(* Logix 5000 project; controller NSH_PLC1 vendor 1 type 14 code 167 rev 32.11; software revision 32.02; part 4 of 12 *)
(* tags used below, declared in another part *)
   H42C : Motor;   // S.Roll
   H42D : Motor;   // Shr.Roll.
   H43A : Motor;   // Aspirator
   H43B : Motor;   // Aspirator
   H49 : Motor;   // Ele.
   H50A : Motor;   // Auger
   H50B : Motor;   // Auger
   M16 : Motor;   // Evo.
   M17 : Motor;   // Evo.
   M18 : Motor;   // Vib.
   M19 : Motor;   // Ele.
   S1 : Motor;   // Vib.
   S10 : Motor;   // Auger
   S13 : Motor;   // Ele.
   S14 : Motor;   // Auger
   S15 : Motor;   // Auger
   S16A : Motor;   // Auger
   S16B : Motor;   // Auger
   S17A : Motor;   // HS Cracker
   S17B : Motor;   // Hard Crkr.
   S17C : Motor;   // Shr.Roll.
   S17D : Motor;   // S.Roll
   S18A : Motor;   // HC Vib.
   S18B : Motor;   // Hard Crkr.
   S18C : Motor;   // Shr.Roll.
   S18D : Motor;   // S.Roll
   S19 : Motor;   // Gry.
   S2 : Motor;   // Ele.
   S20 : Motor;   // Ele.
   S21 : Motor;   // Roll Fdr.
   S22A : Motor;   // HC Vib.
   S22B : Motor;   // Hard Crkr.
   S22C : Motor;   // Shr.Roll.
   S22D : Motor;   // S.Roll
   S23A : Motor;   // HC Vib.
   S23B : Motor;   // Hard Crkr.
   S23C : Motor;   // Shr.Roll.
   S23D : Motor;   // S.Roll
   S24 : Motor;   // Deck
   S25 : Motor;   // Ele.
   S26 : Motor;   // Auger
   S27 : Motor;   // Roll Fdr
   S28A : Motor;   // HC Vib.
   S28B : Motor;   // Hard Crkr.
   S28C : Motor;   // Shr.Roll.
   S28D : Motor;   // S.Roll
   S29A : Motor;   // HC Vib.
   S29B : Motor;   // Hard Crkr.
   S29C : Motor;   // Shr.Roll.
   S29D : Motor;   // S.Roll
   S3 : Motor;   // Auger
   S30 : Motor;   // Ele.
   S31 : Motor;   // Auger
   S32A : Motor;   // HC Vib.
   S32B : Motor;   // Hard Crkr.
   S34 : Motor;   // Deck
   S35 : Motor;   // Ele.
   S36 : Motor;   // Auger
   S38 : Motor;   // Shkr.
   S39 : Motor;   // Ele.
   S41 : Motor;   // Ele.
   S43 : Motor;   // Shkr.
   S44 : Motor;   // Ele.
   S45 : Motor;   // Auger
   S4A : Motor;   // Aspirator
   S4B : Motor;   // Aspirator
   S5A : Motor;   // Aspirator
   S5B : Motor;   // Aspirator
   S6 : Motor;   // Belt
   S7 : Motor;   // Ele.
   S8 : Motor;   // Auger
   S9 : Motor;   // Ele.
(* HullerSheller, continued *)

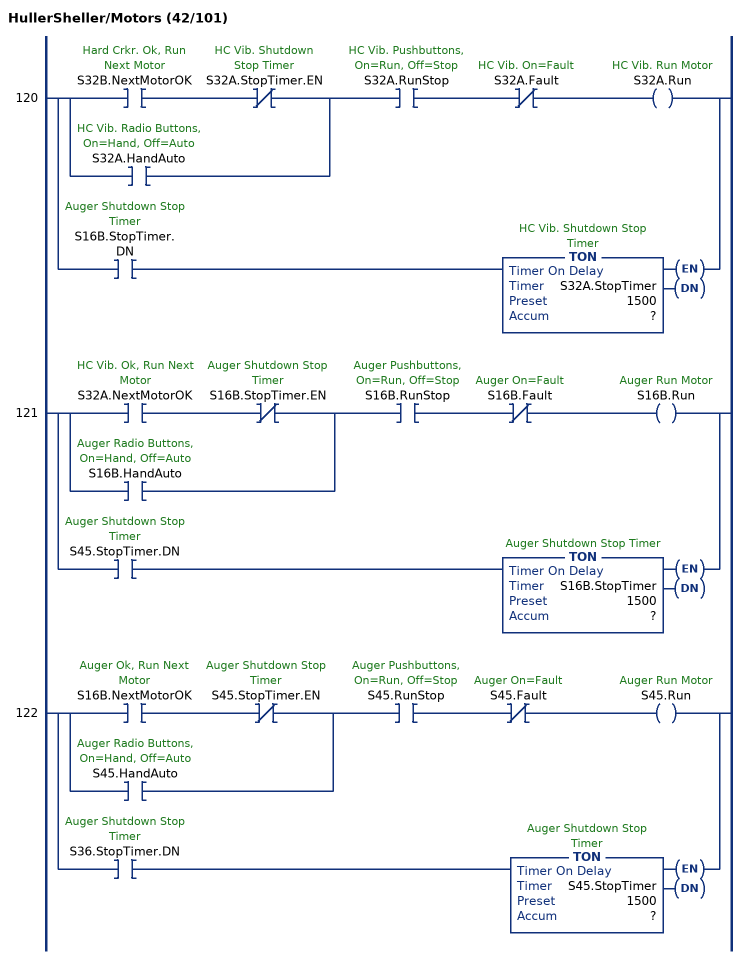
   [picture p66: HullerSheller/Motors rungs 120-122]
   120: [[XIC(S32B.NextMotorOK) XIO(S32A.StopTimer.EN) ,XIC(S32A.HandAuto) ] XIC(S32A.RunStop) XIO(S32A.Fault) OTE(S32A.Run) ,XIC(S16B.StopTimer.DN) TON(S32A.StopTimer,?,?) ];
   121: [[XIC(S32A.NextMotorOK) XIO(S16B.StopTimer.EN) ,XIC(S16B.HandAuto) ] XIC(S16B.RunStop) XIO(S16B.Fault) OTE(S16B.Run) ,XIC(S45.StopTimer.DN) TON(S16B.StopTimer,?,?) ];
   122: [[XIC(S16B.NextMotorOK) XIO(S45.StopTimer.EN) ,XIC(S45.HandAuto) ] XIC(S45.RunStop) XIO(S45.Fault) OTE(S45.Run) ,XIC(S36.StopTimer.DN) TON(S45.StopTimer,?,?) ];
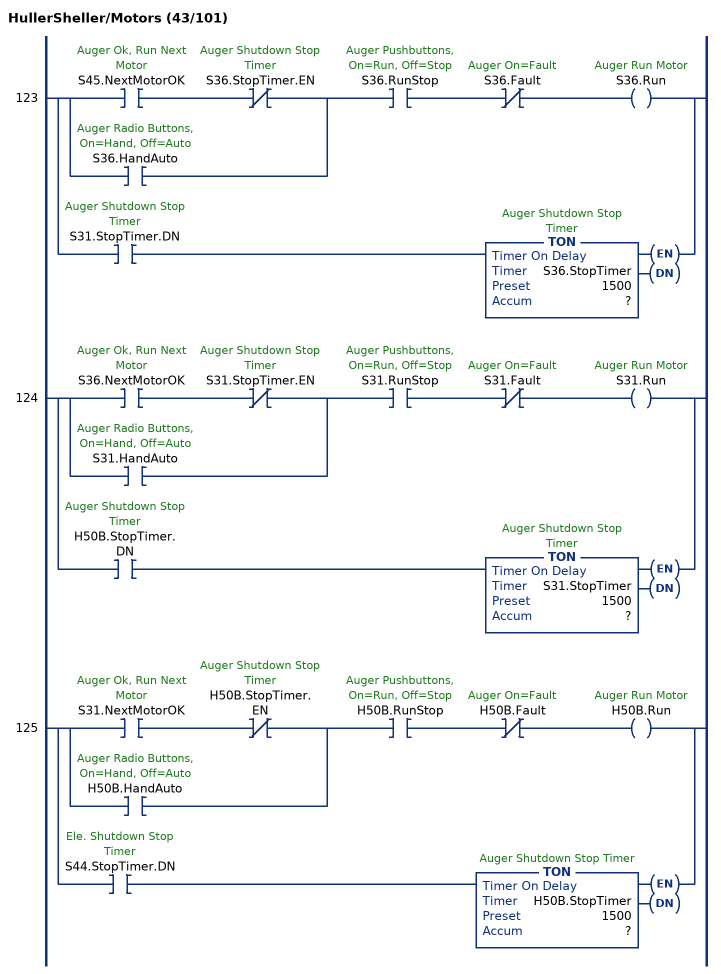
   123: [[XIC(S45.NextMotorOK) XIO(S36.StopTimer.EN) ,XIC(S36.HandAuto) ] XIC(S36.RunStop) XIO(S36.Fault) OTE(S36.Run) ,XIC(S31.StopTimer.DN) TON(S36.StopTimer,?,?) ];
   124: [[XIC(S36.NextMotorOK) XIO(S31.StopTimer.EN) ,XIC(S31.HandAuto) ] XIC(S31.RunStop) XIO(S31.Fault) OTE(S31.Run) ,XIC(H50B.StopTimer.DN) TON(S31.StopTimer,?,?) ];
   125: [[XIC(S31.NextMotorOK) XIO(H50B.StopTimer.EN) ,XIC(H50B.HandAuto) ] XIC(H50B.RunStop) XIO(H50B.Fault) OTE(H50B.Run) ,XIC(S44.StopTimer.DN) TON(H50B.StopTimer,?,?) ];
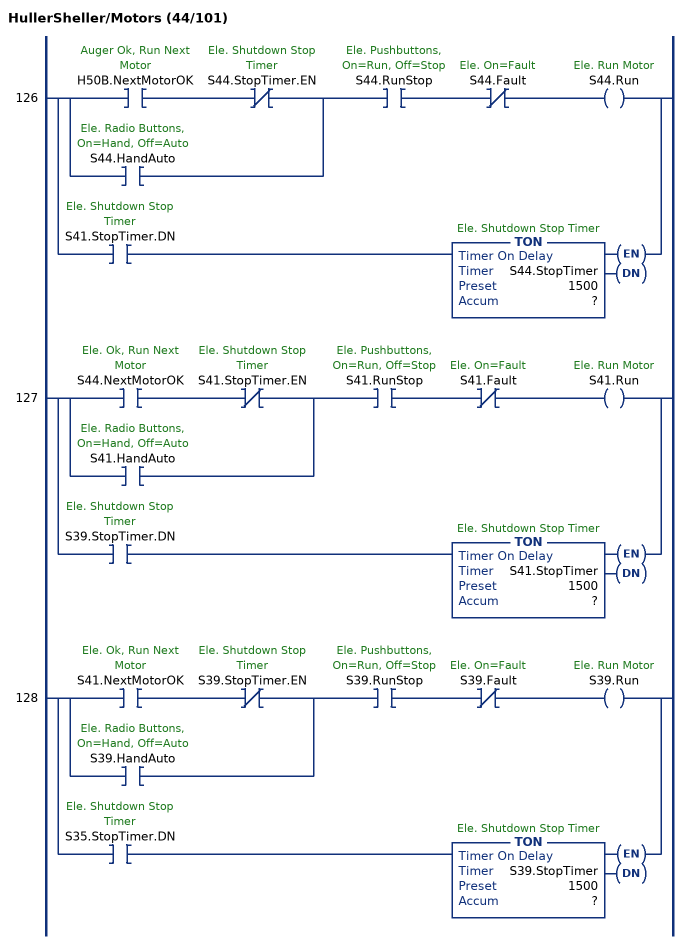
   126: [[XIC(H50B.NextMotorOK) XIO(S44.StopTimer.EN) ,XIC(S44.HandAuto) ] XIC(S44.RunStop) XIO(S44.Fault) OTE(S44.Run) ,XIC(S41.StopTimer.DN) TON(S44.StopTimer,?,?) ];
   127: [[XIC(S44.NextMotorOK) XIO(S41.StopTimer.EN) ,XIC(S41.HandAuto) ] XIC(S41.RunStop) XIO(S41.Fault) OTE(S41.Run) ,XIC(S39.StopTimer.DN) TON(S41.StopTimer,?,?) ];
   128: [[XIC(S41.NextMotorOK) XIO(S39.StopTimer.EN) ,XIC(S39.HandAuto) ] XIC(S39.RunStop) XIO(S39.Fault) OTE(S39.Run) ,XIC(S35.StopTimer.DN) TON(S39.StopTimer,?,?) ];
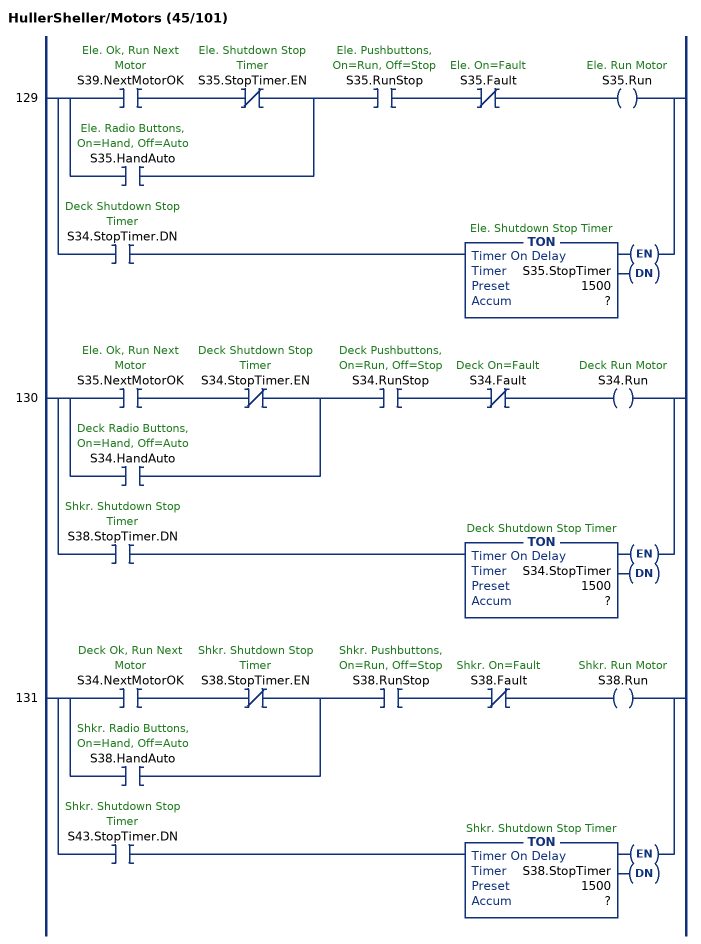
   129: [[XIC(S39.NextMotorOK) XIO(S35.StopTimer.EN) ,XIC(S35.HandAuto) ] XIC(S35.RunStop) XIO(S35.Fault) OTE(S35.Run) ,XIC(S34.StopTimer.DN) TON(S35.StopTimer,?,?) ];
   130: [[XIC(S35.NextMotorOK) XIO(S34.StopTimer.EN) ,XIC(S34.HandAuto) ] XIC(S34.RunStop) XIO(S34.Fault) OTE(S34.Run) ,XIC(S38.StopTimer.DN) TON(S34.StopTimer,?,?) ];
   131: [[XIC(S34.NextMotorOK) XIO(S38.StopTimer.EN) ,XIC(S38.HandAuto) ] XIC(S38.RunStop) XIO(S38.Fault) OTE(S38.Run) ,XIC(S43.StopTimer.DN) TON(S38.StopTimer,?,?) ];
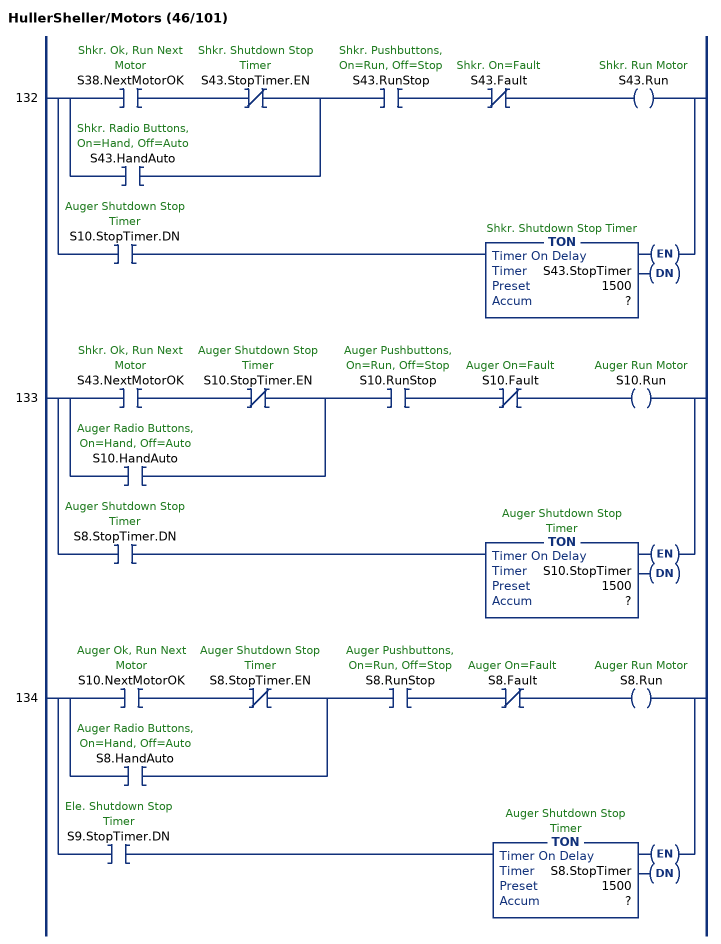
   132: [[XIC(S38.NextMotorOK) XIO(S43.StopTimer.EN) ,XIC(S43.HandAuto) ] XIC(S43.RunStop) XIO(S43.Fault) OTE(S43.Run) ,XIC(S10.StopTimer.DN) TON(S43.StopTimer,?,?) ];
   133: [[XIC(S43.NextMotorOK) XIO(S10.StopTimer.EN) ,XIC(S10.HandAuto) ] XIC(S10.RunStop) XIO(S10.Fault) OTE(S10.Run) ,XIC(S8.StopTimer.DN) TON(S10.StopTimer,?,?) ];
   134: [[XIC(S10.NextMotorOK) XIO(S8.StopTimer.EN) ,XIC(S8.HandAuto) ] XIC(S8.RunStop) XIO(S8.Fault) OTE(S8.Run) ,XIC(S9.StopTimer.DN) TON(S8.StopTimer,?,?) ];
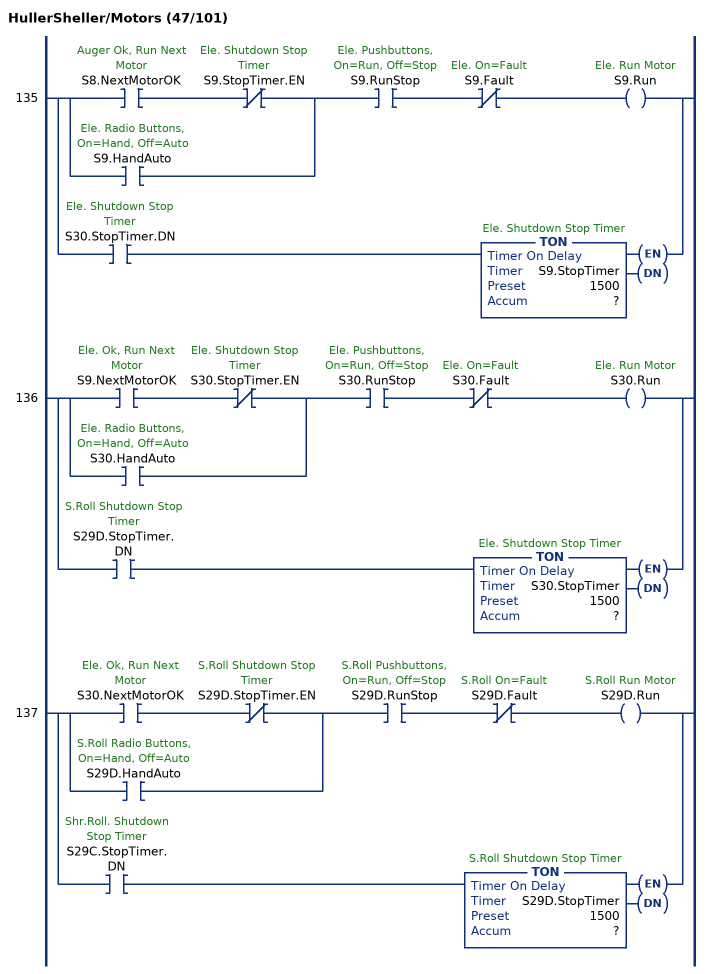
   135: [[XIC(S8.NextMotorOK) XIO(S9.StopTimer.EN) ,XIC(S9.HandAuto) ] XIC(S9.RunStop) XIO(S9.Fault) OTE(S9.Run) ,XIC(S30.StopTimer.DN) TON(S9.StopTimer,?,?) ];
   136: [[XIC(S9.NextMotorOK) XIO(S30.StopTimer.EN) ,XIC(S30.HandAuto) ] XIC(S30.RunStop) XIO(S30.Fault) OTE(S30.Run) ,XIC(S29D.StopTimer.DN) TON(S30.StopTimer,?,?) ];
   137: [[XIC(S30.NextMotorOK) XIO(S29D.StopTimer.EN) ,XIC(S29D.HandAuto) ] XIC(S29D.RunStop) XIO(S29D.Fault) OTE(S29D.Run) ,XIC(S29C.StopTimer.DN) TON(S29D.StopTimer,?,?) ];
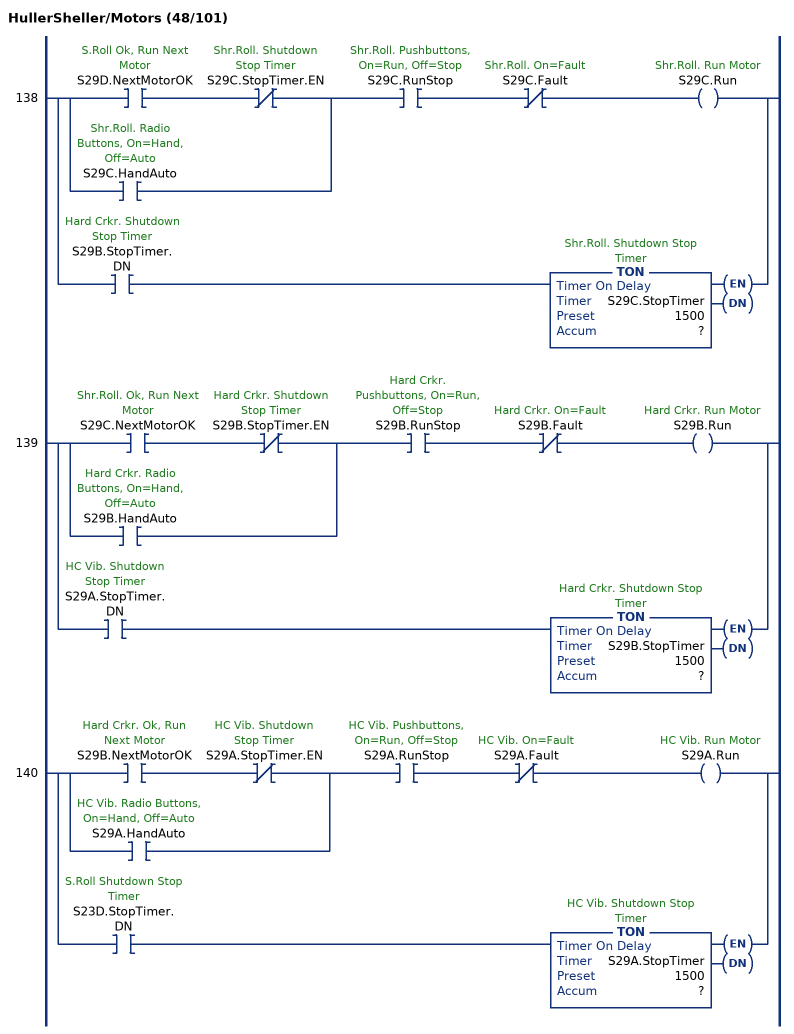
   138: [[XIC(S29D.NextMotorOK) XIO(S29C.StopTimer.EN) ,XIC(S29C.HandAuto) ] XIC(S29C.RunStop) XIO(S29C.Fault) OTE(S29C.Run) ,XIC(S29B.StopTimer.DN) TON(S29C.StopTimer,?,?) ];
   139: [[XIC(S29C.NextMotorOK) XIO(S29B.StopTimer.EN) ,XIC(S29B.HandAuto) ] XIC(S29B.RunStop) XIO(S29B.Fault) OTE(S29B.Run) ,XIC(S29A.StopTimer.DN) TON(S29B.StopTimer,?,?) ];
   140: [[XIC(S29B.NextMotorOK) XIO(S29A.StopTimer.EN) ,XIC(S29A.HandAuto) ] XIC(S29A.RunStop) XIO(S29A.Fault) OTE(S29A.Run) ,XIC(S23D.StopTimer.DN) TON(S29A.StopTimer,?,?) ];
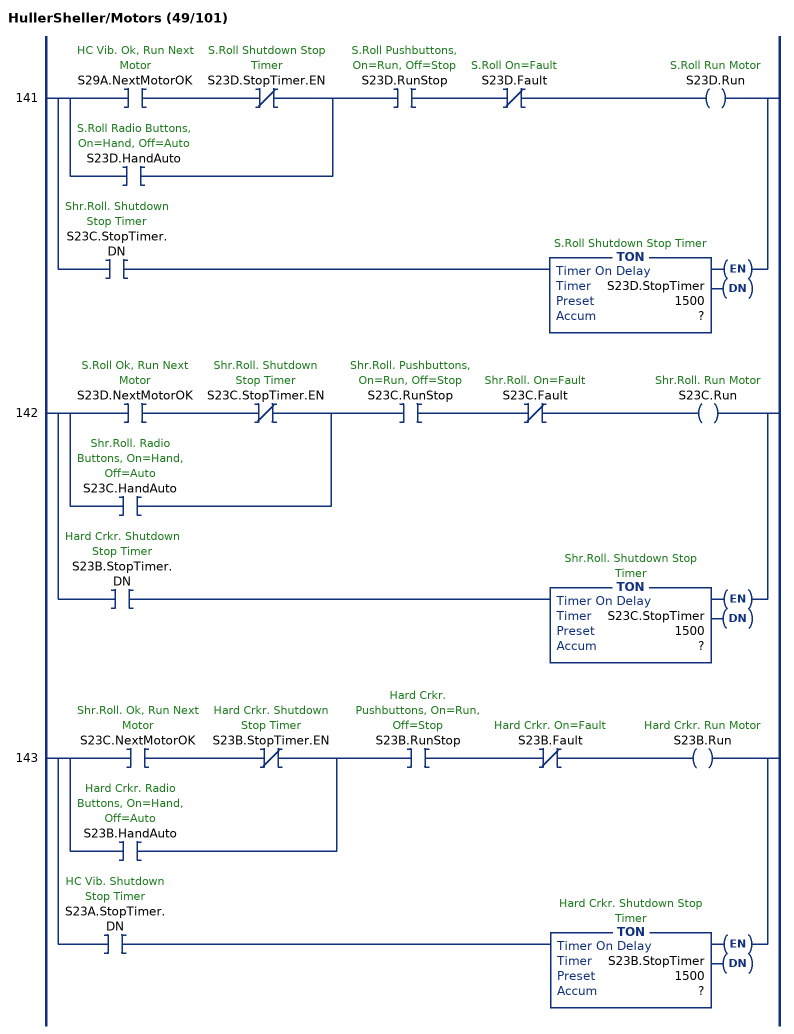
   141: [[XIC(S29A.NextMotorOK) XIO(S23D.StopTimer.EN) ,XIC(S23D.HandAuto) ] XIC(S23D.RunStop) XIO(S23D.Fault) OTE(S23D.Run) ,XIC(S23C.StopTimer.DN) TON(S23D.StopTimer,?,?) ];
   142: [[XIC(S23D.NextMotorOK) XIO(S23C.StopTimer.EN) ,XIC(S23C.HandAuto) ] XIC(S23C.RunStop) XIO(S23C.Fault) OTE(S23C.Run) ,XIC(S23B.StopTimer.DN) TON(S23C.StopTimer,?,?) ];
   143: [[XIC(S23C.NextMotorOK) XIO(S23B.StopTimer.EN) ,XIC(S23B.HandAuto) ] XIC(S23B.RunStop) XIO(S23B.Fault) OTE(S23B.Run) ,XIC(S23A.StopTimer.DN) TON(S23B.StopTimer,?,?) ];
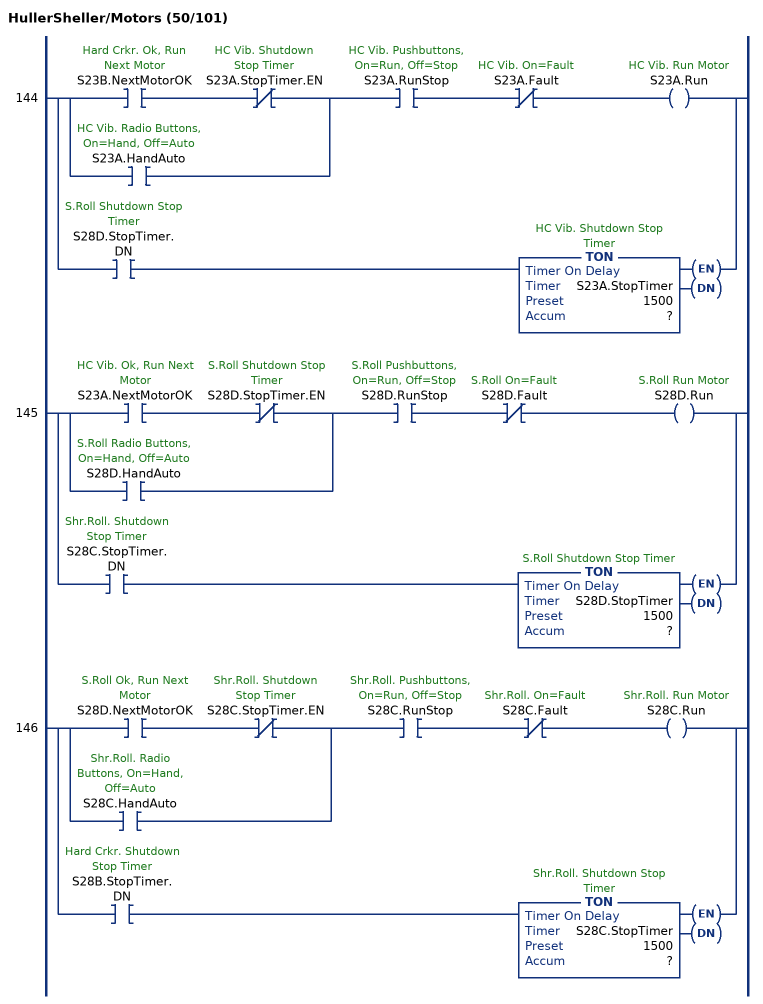
   144: [[XIC(S23B.NextMotorOK) XIO(S23A.StopTimer.EN) ,XIC(S23A.HandAuto) ] XIC(S23A.RunStop) XIO(S23A.Fault) OTE(S23A.Run) ,XIC(S28D.StopTimer.DN) TON(S23A.StopTimer,?,?) ];
   145: [[XIC(S23A.NextMotorOK) XIO(S28D.StopTimer.EN) ,XIC(S28D.HandAuto) ] XIC(S28D.RunStop) XIO(S28D.Fault) OTE(S28D.Run) ,XIC(S28C.StopTimer.DN) TON(S28D.StopTimer,?,?) ];
   146: [[XIC(S28D.NextMotorOK) XIO(S28C.StopTimer.EN) ,XIC(S28C.HandAuto) ] XIC(S28C.RunStop) XIO(S28C.Fault) OTE(S28C.Run) ,XIC(S28B.StopTimer.DN) TON(S28C.StopTimer,?,?) ];
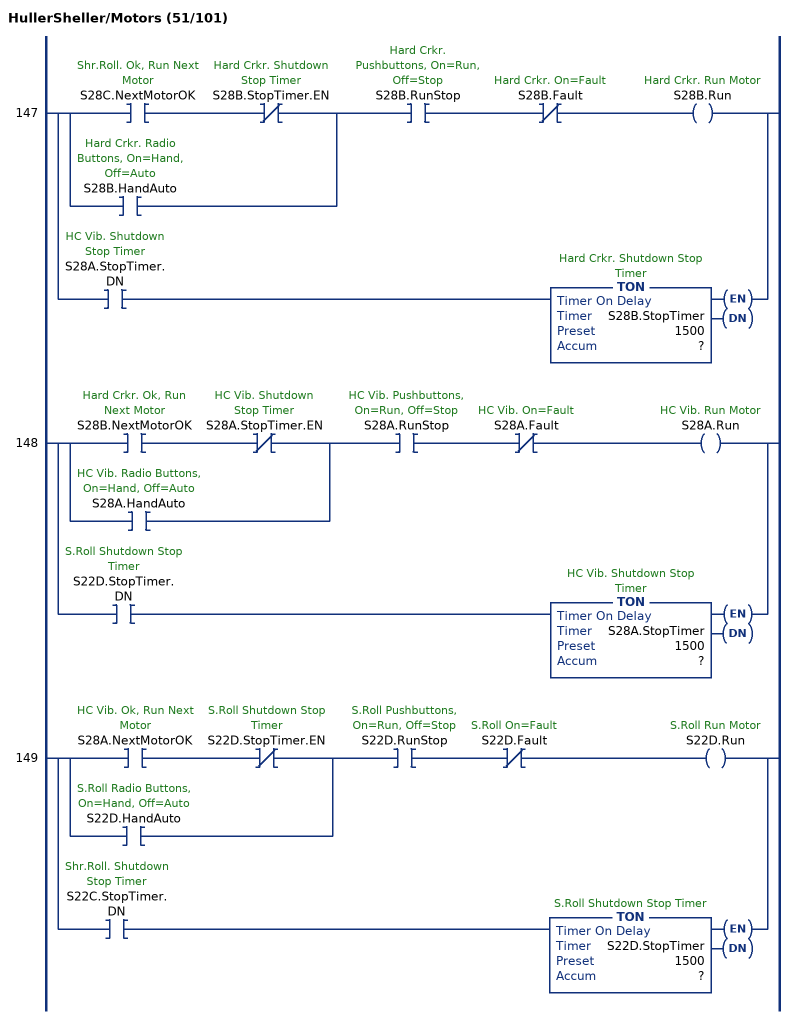
   147: [[XIC(S28C.NextMotorOK) XIO(S28B.StopTimer.EN) ,XIC(S28B.HandAuto) ] XIC(S28B.RunStop) XIO(S28B.Fault) OTE(S28B.Run) ,XIC(S28A.StopTimer.DN) TON(S28B.StopTimer,?,?) ];
   148: [[XIC(S28B.NextMotorOK) XIO(S28A.StopTimer.EN) ,XIC(S28A.HandAuto) ] XIC(S28A.RunStop) XIO(S28A.Fault) OTE(S28A.Run) ,XIC(S22D.StopTimer.DN) TON(S28A.StopTimer,?,?) ];
   149: [[XIC(S28A.NextMotorOK) XIO(S22D.StopTimer.EN) ,XIC(S22D.HandAuto) ] XIC(S22D.RunStop) XIO(S22D.Fault) OTE(S22D.Run) ,XIC(S22C.StopTimer.DN) TON(S22D.StopTimer,?,?) ];
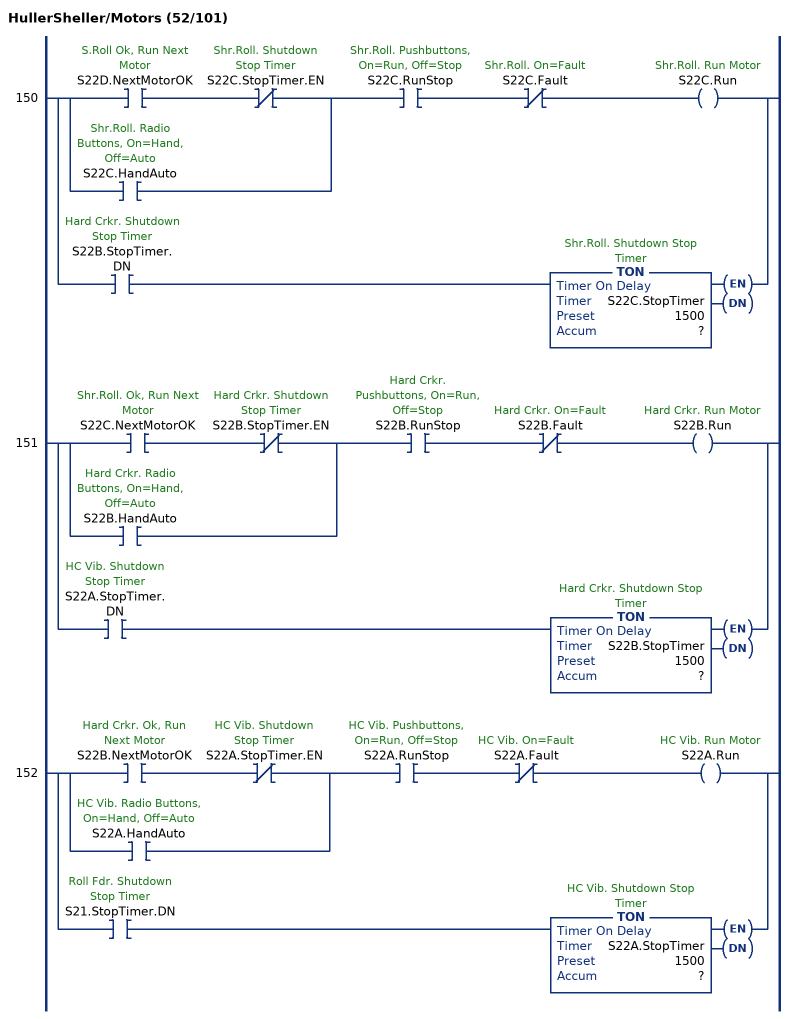
   150: [[XIC(S22D.NextMotorOK) XIO(S22C.StopTimer.EN) ,XIC(S22C.HandAuto) ] XIC(S22C.RunStop) XIO(S22C.Fault) OTE(S22C.Run) ,XIC(S22B.StopTimer.DN) TON(S22C.StopTimer,?,?) ];
   151: [[XIC(S22C.NextMotorOK) XIO(S22B.StopTimer.EN) ,XIC(S22B.HandAuto) ] XIC(S22B.RunStop) XIO(S22B.Fault) OTE(S22B.Run) ,XIC(S22A.StopTimer.DN) TON(S22B.StopTimer,?,?) ];
   152: [[XIC(S22B.NextMotorOK) XIO(S22A.StopTimer.EN) ,XIC(S22A.HandAuto) ] XIC(S22A.RunStop) XIO(S22A.Fault) OTE(S22A.Run) ,XIC(S21.StopTimer.DN) TON(S22A.StopTimer,?,?) ];
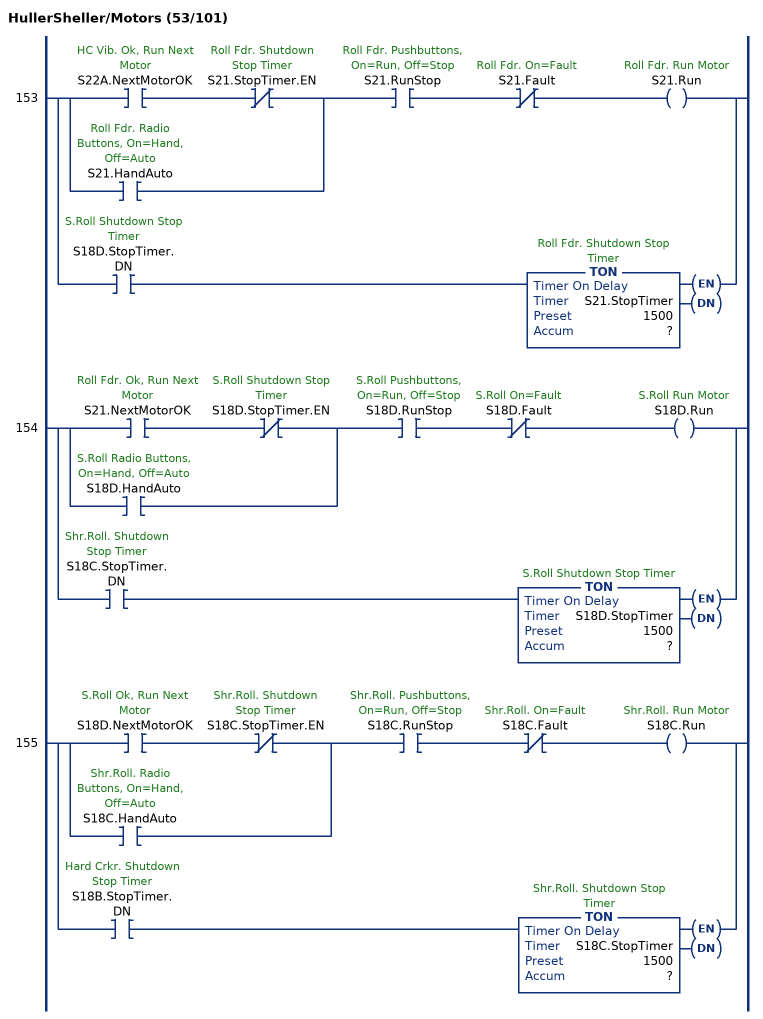
   153: [[XIC(S22A.NextMotorOK) XIO(S21.StopTimer.EN) ,XIC(S21.HandAuto) ] XIC(S21.RunStop) XIO(S21.Fault) OTE(S21.Run) ,XIC(S18D.StopTimer.DN) TON(S21.StopTimer,?,?) ];
   154: [[XIC(S21.NextMotorOK) XIO(S18D.StopTimer.EN) ,XIC(S18D.HandAuto) ] XIC(S18D.RunStop) XIO(S18D.Fault) OTE(S18D.Run) ,XIC(S18C.StopTimer.DN) TON(S18D.StopTimer,?,?) ];
   155: [[XIC(S18D.NextMotorOK) XIO(S18C.StopTimer.EN) ,XIC(S18C.HandAuto) ] XIC(S18C.RunStop) XIO(S18C.Fault) OTE(S18C.Run) ,XIC(S18B.StopTimer.DN) TON(S18C.StopTimer,?,?) ];
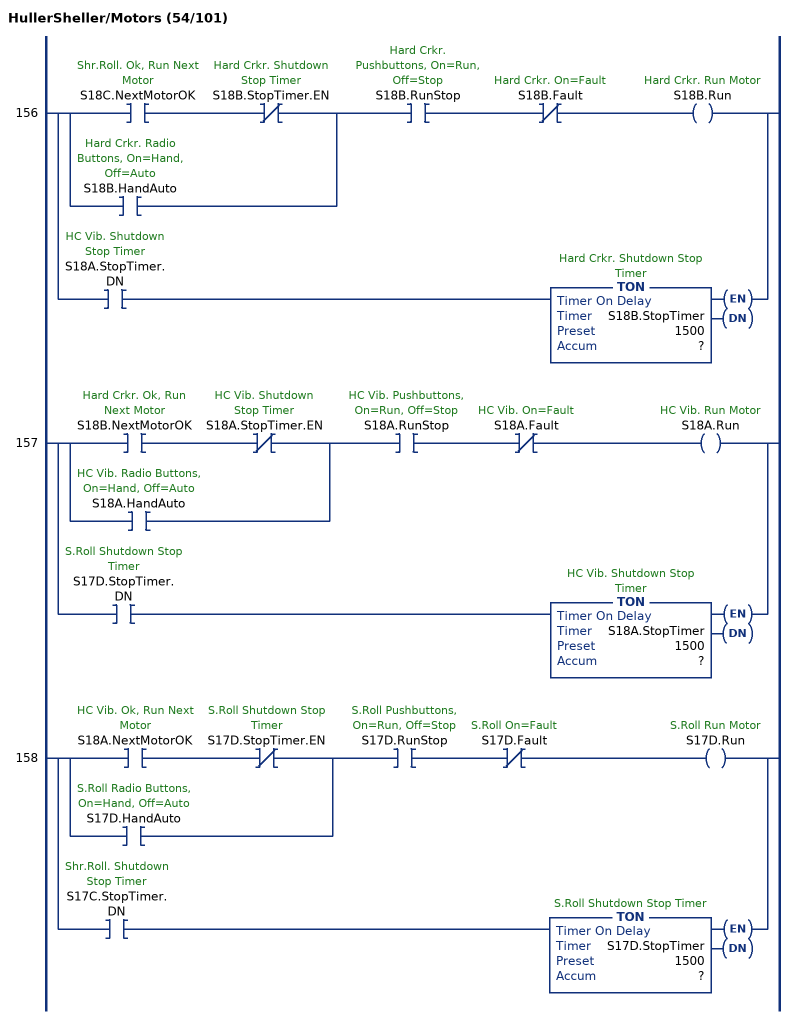
   156: [[XIC(S18C.NextMotorOK) XIO(S18B.StopTimer.EN) ,XIC(S18B.HandAuto) ] XIC(S18B.RunStop) XIO(S18B.Fault) OTE(S18B.Run) ,XIC(S18A.StopTimer.DN) TON(S18B.StopTimer,?,?) ];
   157: [[XIC(S18B.NextMotorOK) XIO(S18A.StopTimer.EN) ,XIC(S18A.HandAuto) ] XIC(S18A.RunStop) XIO(S18A.Fault) OTE(S18A.Run) ,XIC(S17D.StopTimer.DN) TON(S18A.StopTimer,?,?) ];
   158: [[XIC(S18A.NextMotorOK) XIO(S17D.StopTimer.EN) ,XIC(S17D.HandAuto) ] XIC(S17D.RunStop) XIO(S17D.Fault) OTE(S17D.Run) ,XIC(S17C.StopTimer.DN) TON(S17D.StopTimer,?,?) ];
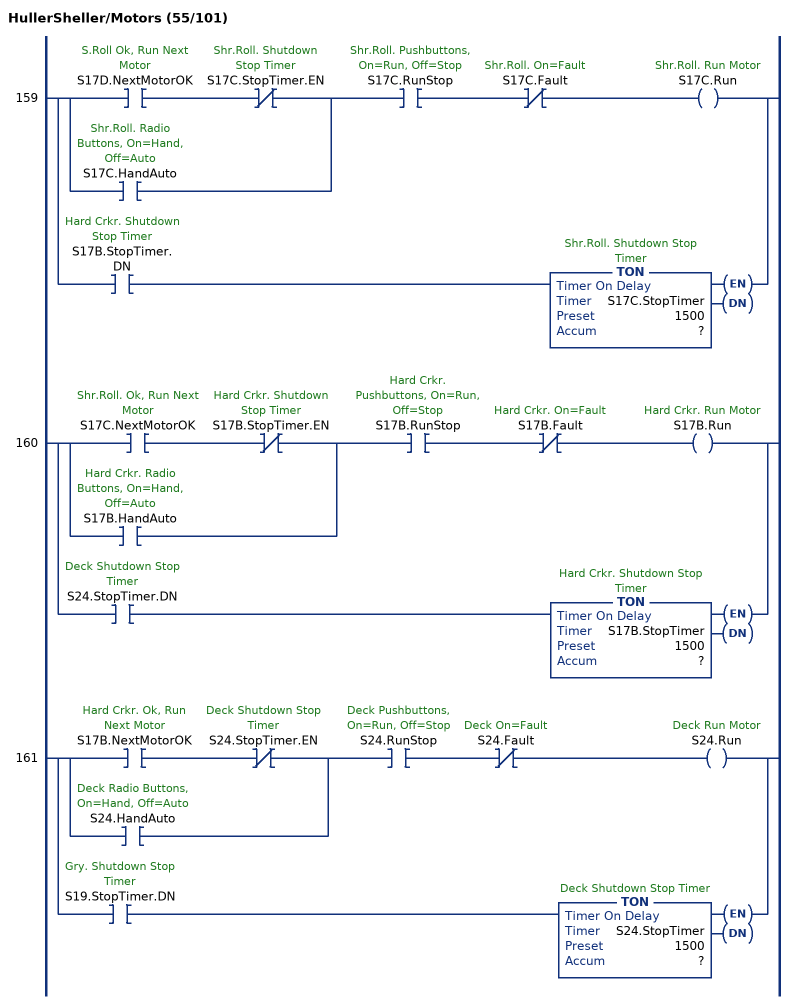
   159: [[XIC(S17D.NextMotorOK) XIO(S17C.StopTimer.EN) ,XIC(S17C.HandAuto) ] XIC(S17C.RunStop) XIO(S17C.Fault) OTE(S17C.Run) ,XIC(S17B.StopTimer.DN) TON(S17C.StopTimer,?,?) ];
   160: [[XIC(S17C.NextMotorOK) XIO(S17B.StopTimer.EN) ,XIC(S17B.HandAuto) ] XIC(S17B.RunStop) XIO(S17B.Fault) OTE(S17B.Run) ,XIC(S24.StopTimer.DN) TON(S17B.StopTimer,?,?) ];
   161: [[XIC(S17B.NextMotorOK) XIO(S24.StopTimer.EN) ,XIC(S24.HandAuto) ] XIC(S24.RunStop) XIO(S24.Fault) OTE(S24.Run) ,XIC(S19.StopTimer.DN) TON(S24.StopTimer,?,?) ];
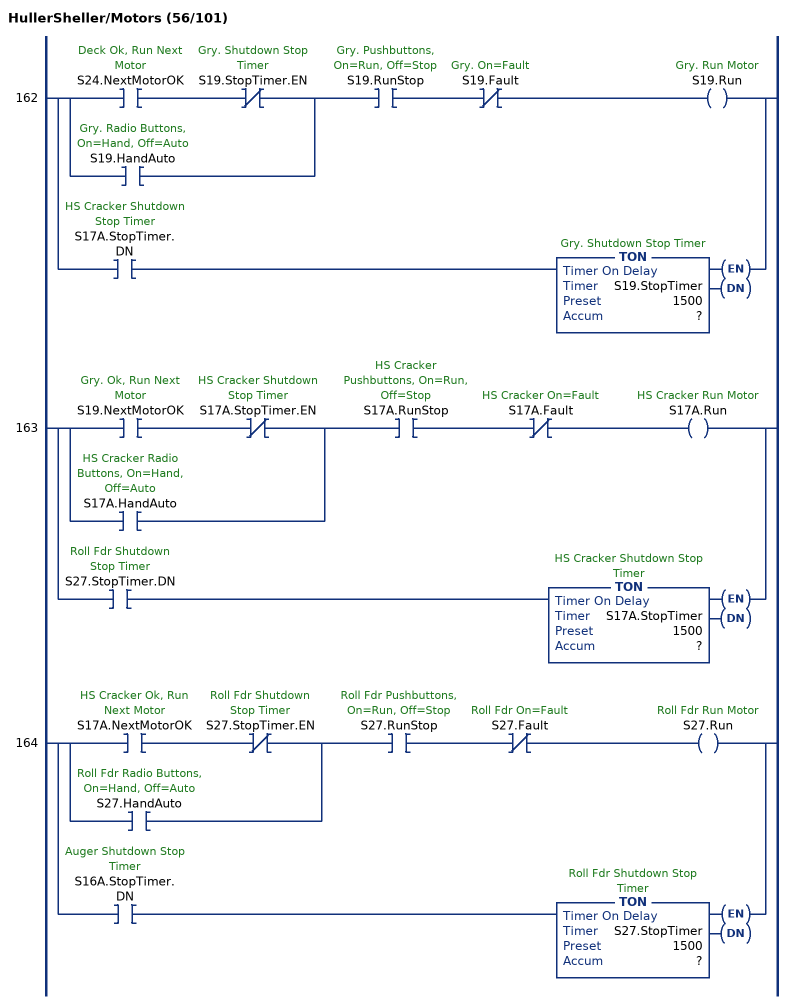
   162: [[XIC(S24.NextMotorOK) XIO(S19.StopTimer.EN) ,XIC(S19.HandAuto) ] XIC(S19.RunStop) XIO(S19.Fault) OTE(S19.Run) ,XIC(S17A.StopTimer.DN) TON(S19.StopTimer,?,?) ];
   163: [[XIC(S19.NextMotorOK) XIO(S17A.StopTimer.EN) ,XIC(S17A.HandAuto) ] XIC(S17A.RunStop) XIO(S17A.Fault) OTE(S17A.Run) ,XIC(S27.StopTimer.DN) TON(S17A.StopTimer,?,?) ];
   164: [[XIC(S17A.NextMotorOK) XIO(S27.StopTimer.EN) ,XIC(S27.HandAuto) ] XIC(S27.RunStop) XIO(S27.Fault) OTE(S27.Run) ,XIC(S16A.StopTimer.DN) TON(S27.StopTimer,?,?) ];
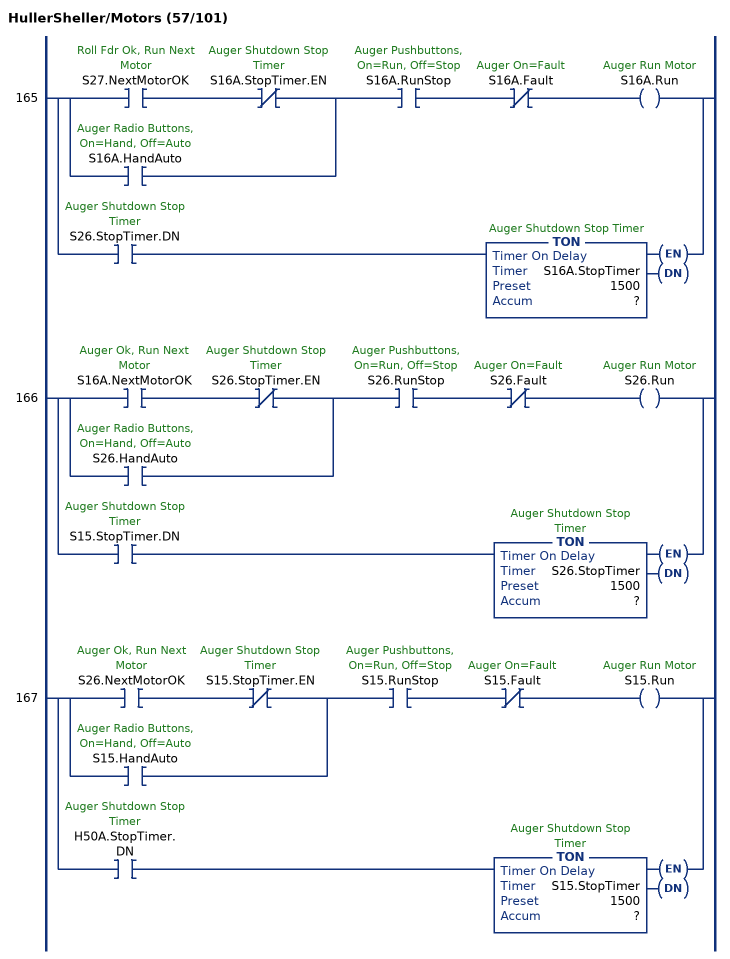
   165: [[XIC(S27.NextMotorOK) XIO(S16A.StopTimer.EN) ,XIC(S16A.HandAuto) ] XIC(S16A.RunStop) XIO(S16A.Fault) OTE(S16A.Run) ,XIC(S26.StopTimer.DN) TON(S16A.StopTimer,?,?) ];
   166: [[XIC(S16A.NextMotorOK) XIO(S26.StopTimer.EN) ,XIC(S26.HandAuto) ] XIC(S26.RunStop) XIO(S26.Fault) OTE(S26.Run) ,XIC(S15.StopTimer.DN) TON(S26.StopTimer,?,?) ];
   167: [[XIC(S26.NextMotorOK) XIO(S15.StopTimer.EN) ,XIC(S15.HandAuto) ] XIC(S15.RunStop) XIO(S15.Fault) OTE(S15.Run) ,XIC(H50A.StopTimer.DN) TON(S15.StopTimer,?,?) ];
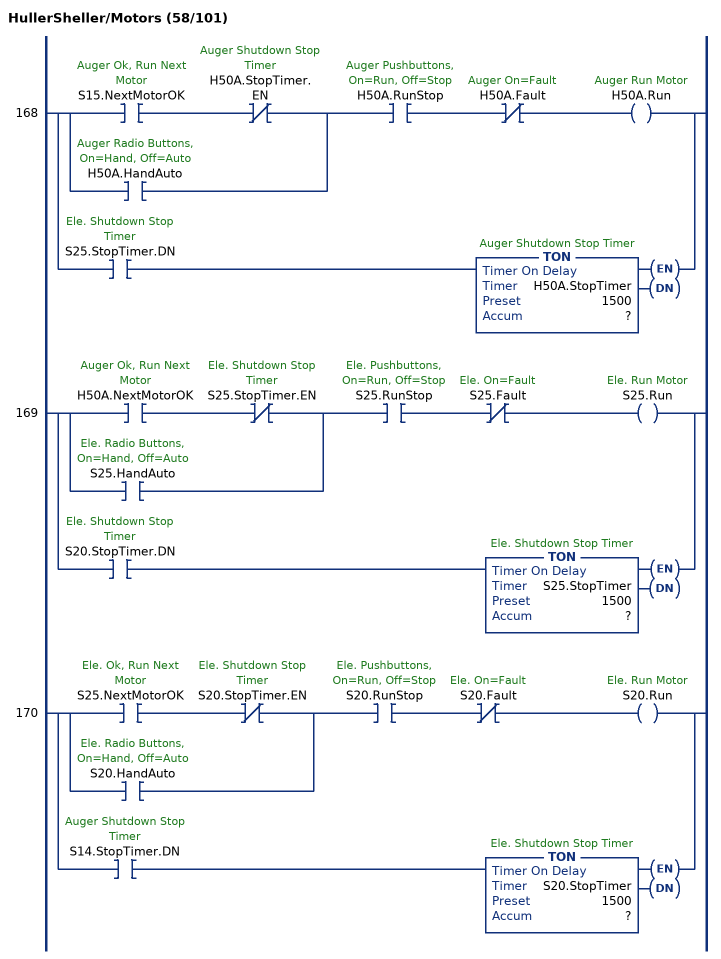
   168: [[XIC(S15.NextMotorOK) XIO(H50A.StopTimer.EN) ,XIC(H50A.HandAuto) ] XIC(H50A.RunStop) XIO(H50A.Fault) OTE(H50A.Run) ,XIC(S25.StopTimer.DN) TON(H50A.StopTimer,?,?) ];
   169: [[XIC(H50A.NextMotorOK) XIO(S25.StopTimer.EN) ,XIC(S25.HandAuto) ] XIC(S25.RunStop) XIO(S25.Fault) OTE(S25.Run) ,XIC(S20.StopTimer.DN) TON(S25.StopTimer,?,?) ];
   170: [[XIC(S25.NextMotorOK) XIO(S20.StopTimer.EN) ,XIC(S20.HandAuto) ] XIC(S20.RunStop) XIO(S20.Fault) OTE(S20.Run) ,XIC(S14.StopTimer.DN) TON(S20.StopTimer,?,?) ];
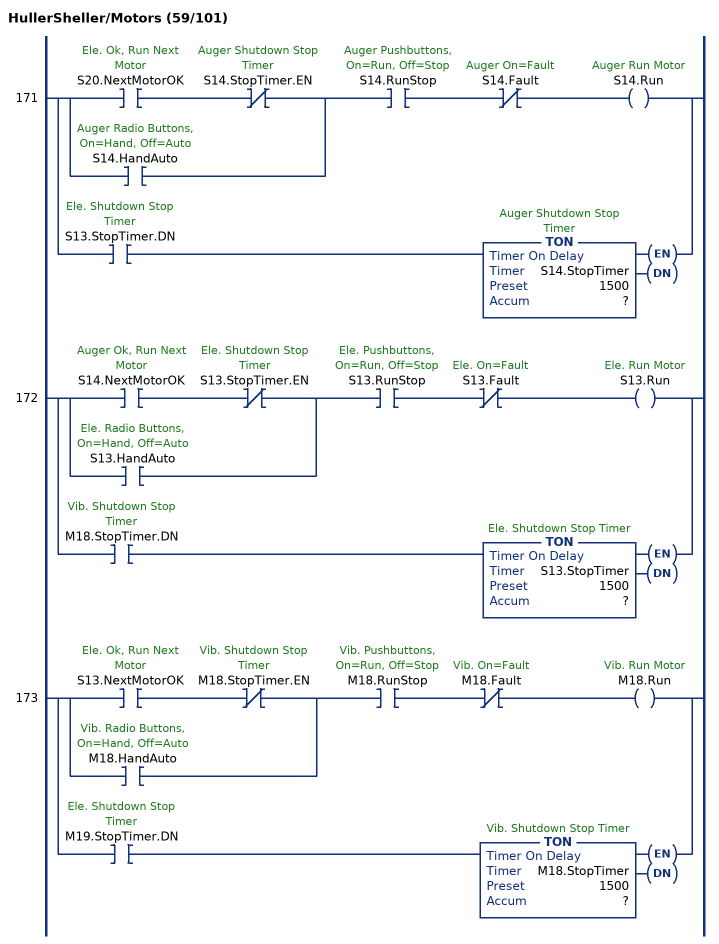
   171: [[XIC(S20.NextMotorOK) XIO(S14.StopTimer.EN) ,XIC(S14.HandAuto) ] XIC(S14.RunStop) XIO(S14.Fault) OTE(S14.Run) ,XIC(S13.StopTimer.DN) TON(S14.StopTimer,?,?) ];
   172: [[XIC(S14.NextMotorOK) XIO(S13.StopTimer.EN) ,XIC(S13.HandAuto) ] XIC(S13.RunStop) XIO(S13.Fault) OTE(S13.Run) ,XIC(M18.StopTimer.DN) TON(S13.StopTimer,?,?) ];
   173: [[XIC(S13.NextMotorOK) XIO(M18.StopTimer.EN) ,XIC(M18.HandAuto) ] XIC(M18.RunStop) XIO(M18.Fault) OTE(M18.Run) ,XIC(M19.StopTimer.DN) TON(M18.StopTimer,?,?) ];
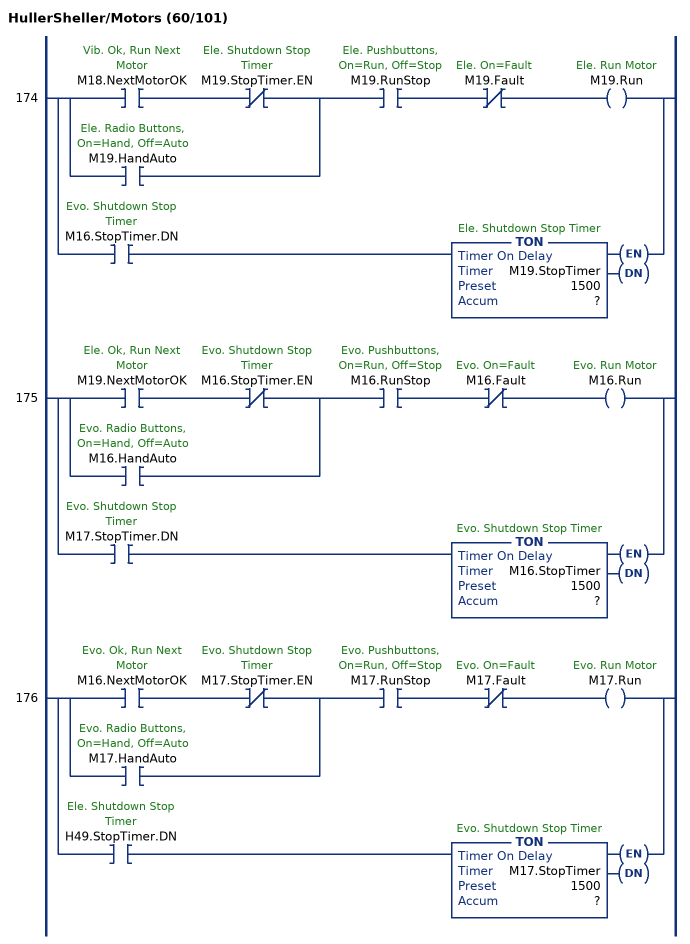
   174: [[XIC(M18.NextMotorOK) XIO(M19.StopTimer.EN) ,XIC(M19.HandAuto) ] XIC(M19.RunStop) XIO(M19.Fault) OTE(M19.Run) ,XIC(M16.StopTimer.DN) TON(M19.StopTimer,?,?) ];
   175: [[XIC(M19.NextMotorOK) XIO(M16.StopTimer.EN) ,XIC(M16.HandAuto) ] XIC(M16.RunStop) XIO(M16.Fault) OTE(M16.Run) ,XIC(M17.StopTimer.DN) TON(M16.StopTimer,?,?) ];
   176: [[XIC(M16.NextMotorOK) XIO(M17.StopTimer.EN) ,XIC(M17.HandAuto) ] XIC(M17.RunStop) XIO(M17.Fault) OTE(M17.Run) ,XIC(H49.StopTimer.DN) TON(M17.StopTimer,?,?) ];
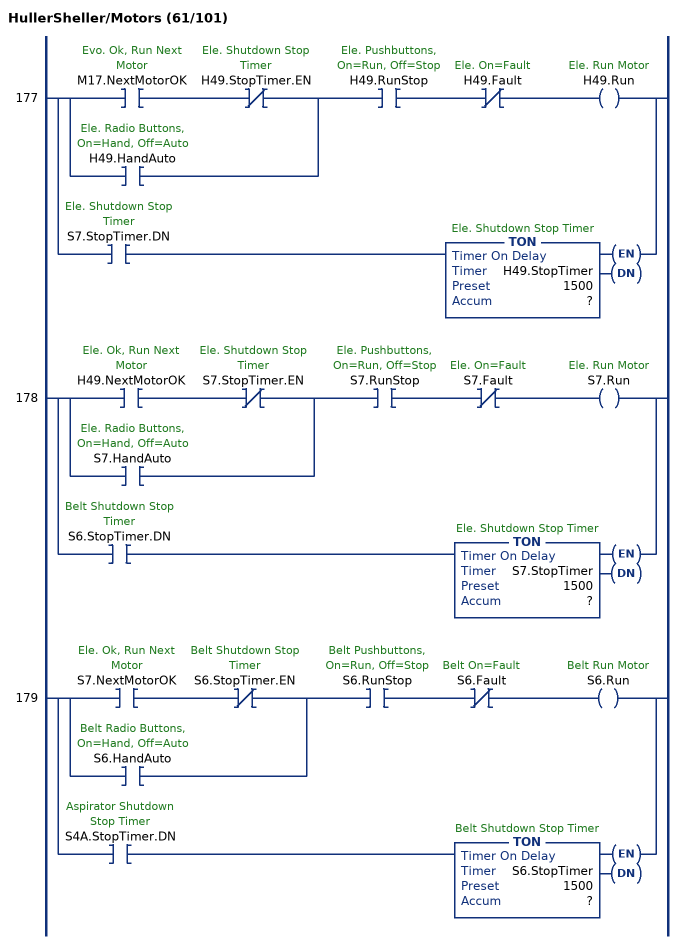
   177: [[XIC(M17.NextMotorOK) XIO(H49.StopTimer.EN) ,XIC(H49.HandAuto) ] XIC(H49.RunStop) XIO(H49.Fault) OTE(H49.Run) ,XIC(S7.StopTimer.DN) TON(H49.StopTimer,?,?) ];
   178: [[XIC(H49.NextMotorOK) XIO(S7.StopTimer.EN) ,XIC(S7.HandAuto) ] XIC(S7.RunStop) XIO(S7.Fault) OTE(S7.Run) ,XIC(S6.StopTimer.DN) TON(S7.StopTimer,?,?) ];
   179: [[XIC(S7.NextMotorOK) XIO(S6.StopTimer.EN) ,XIC(S6.HandAuto) ] XIC(S6.RunStop) XIO(S6.Fault) OTE(S6.Run) ,XIC(S4A.StopTimer.DN) TON(S6.StopTimer,?,?) ];
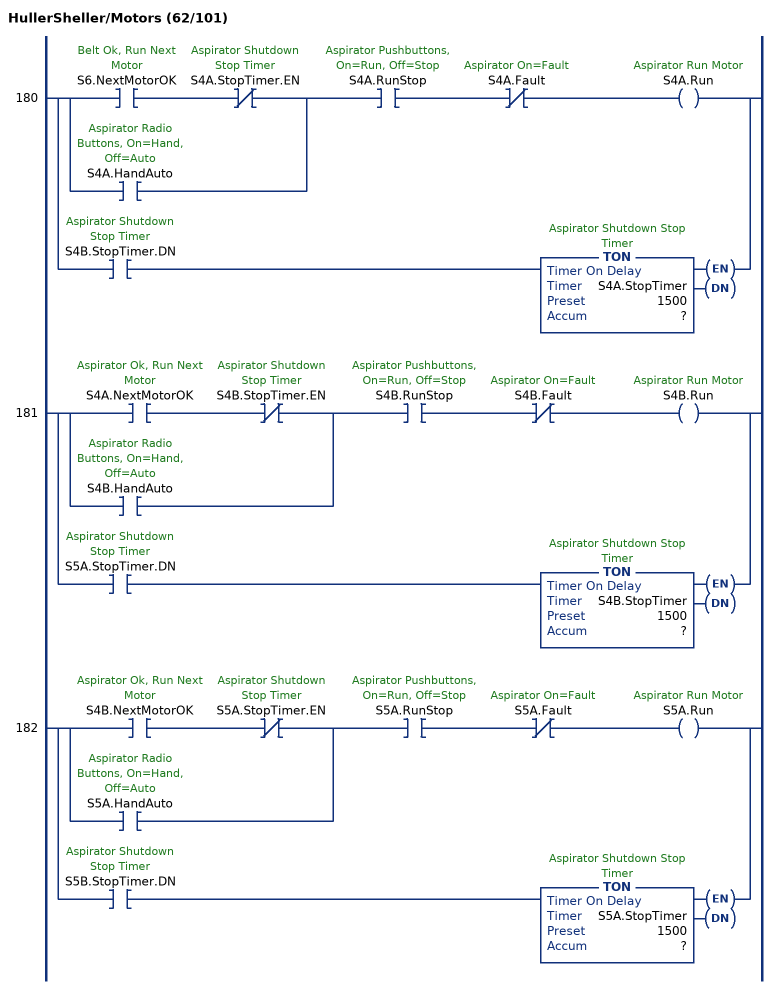
   180: [[XIC(S6.NextMotorOK) XIO(S4A.StopTimer.EN) ,XIC(S4A.HandAuto) ] XIC(S4A.RunStop) XIO(S4A.Fault) OTE(S4A.Run) ,XIC(S4B.StopTimer.DN) TON(S4A.StopTimer,?,?) ];
   181: [[XIC(S4A.NextMotorOK) XIO(S4B.StopTimer.EN) ,XIC(S4B.HandAuto) ] XIC(S4B.RunStop) XIO(S4B.Fault) OTE(S4B.Run) ,XIC(S5A.StopTimer.DN) TON(S4B.StopTimer,?,?) ];
   182: [[XIC(S4B.NextMotorOK) XIO(S5A.StopTimer.EN) ,XIC(S5A.HandAuto) ] XIC(S5A.RunStop) XIO(S5A.Fault) OTE(S5A.Run) ,XIC(S5B.StopTimer.DN) TON(S5A.StopTimer,?,?) ];
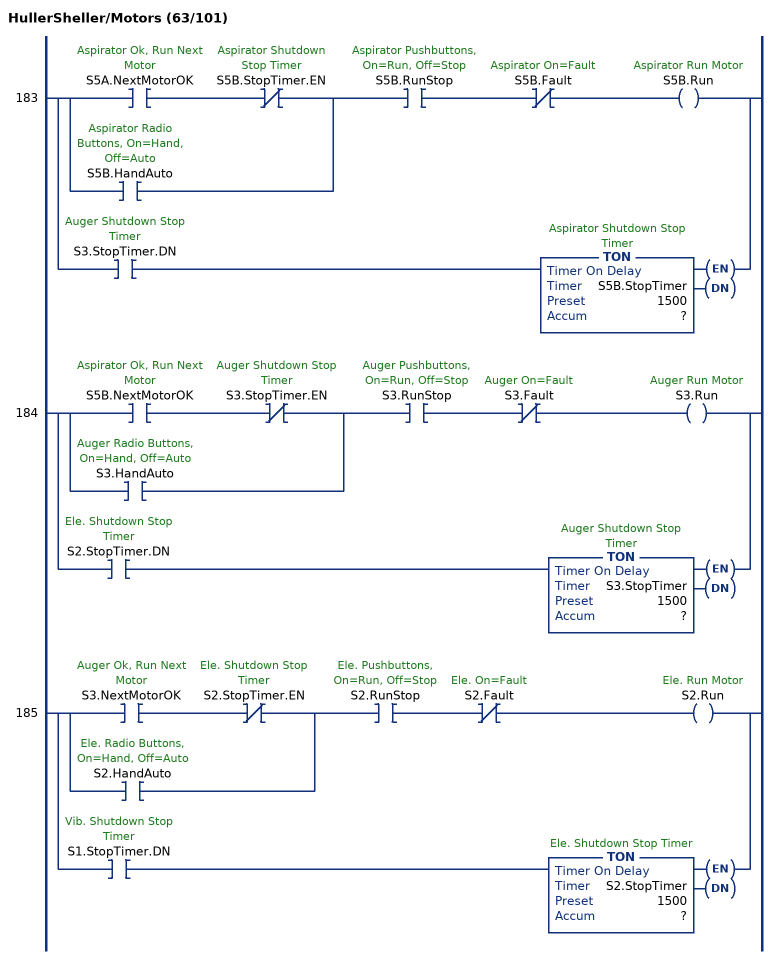
   183: [[XIC(S5A.NextMotorOK) XIO(S5B.StopTimer.EN) ,XIC(S5B.HandAuto) ] XIC(S5B.RunStop) XIO(S5B.Fault) OTE(S5B.Run) ,XIC(S3.StopTimer.DN) TON(S5B.StopTimer,?,?) ];
   184: [[XIC(S5B.NextMotorOK) XIO(S3.StopTimer.EN) ,XIC(S3.HandAuto) ] XIC(S3.RunStop) XIO(S3.Fault) OTE(S3.Run) ,XIC(S2.StopTimer.DN) TON(S3.StopTimer,?,?) ];
   185: [[XIC(S3.NextMotorOK) XIO(S2.StopTimer.EN) ,XIC(S2.HandAuto) ] XIC(S2.RunStop) XIO(S2.Fault) OTE(S2.Run) ,XIC(S1.StopTimer.DN) TON(S2.StopTimer,?,?) ];
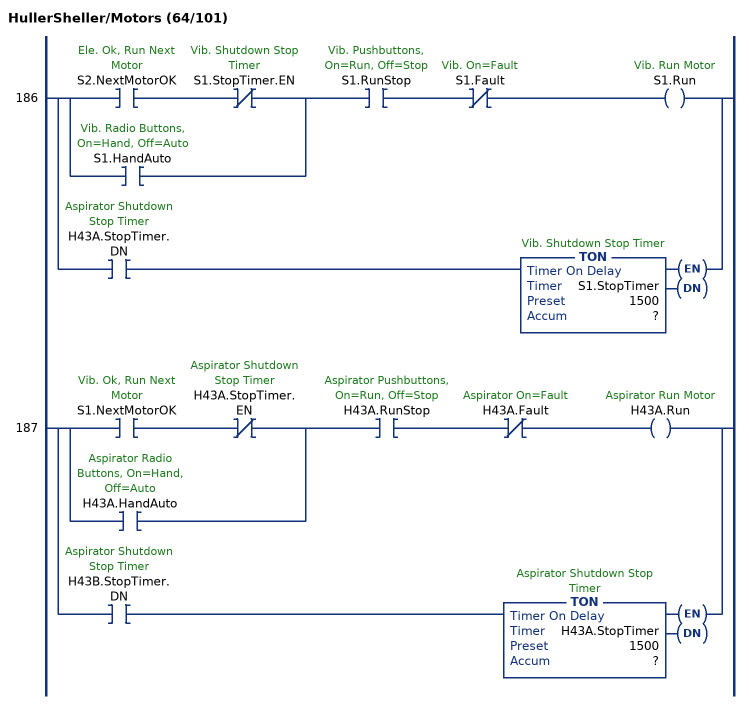
   186: [[XIC(S2.NextMotorOK) XIO(S1.StopTimer.EN) ,XIC(S1.HandAuto) ] XIC(S1.RunStop) XIO(S1.Fault) OTE(S1.Run) ,XIC(H43A.StopTimer.DN) TON(S1.StopTimer,?,?) ];
   187: [[XIC(S1.NextMotorOK) XIO(H43A.StopTimer.EN) ,XIC(H43A.HandAuto) ] XIC(H43A.RunStop) XIO(H43A.Fault) OTE(H43A.Run) ,XIC(H43B.StopTimer.DN) TON(H43A.StopTimer,?,?) ];
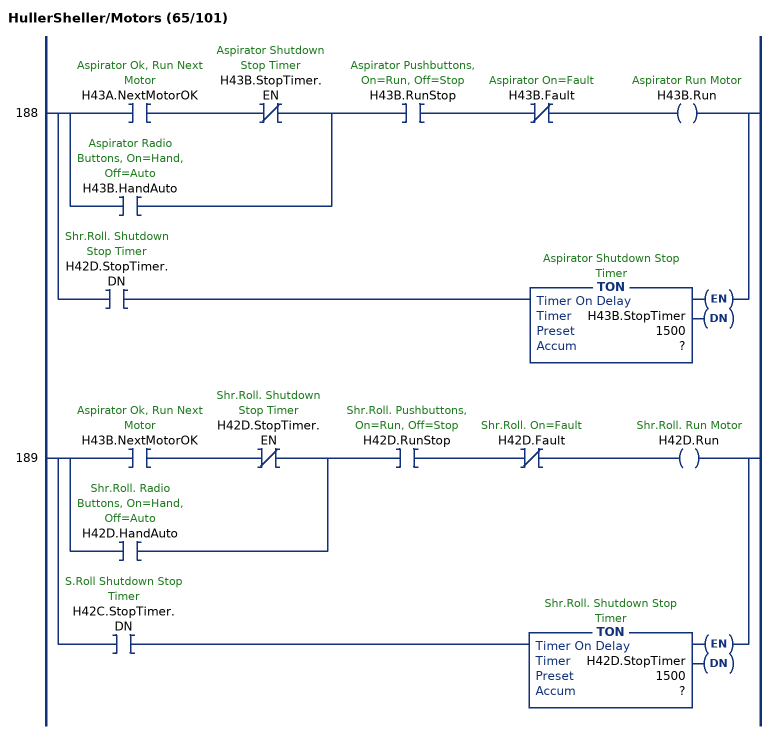
   188: [[XIC(H43A.NextMotorOK) XIO(H43B.StopTimer.EN) ,XIC(H43B.HandAuto) ] XIC(H43B.RunStop) XIO(H43B.Fault) OTE(H43B.Run) ,XIC(H42D.StopTimer.DN) TON(H43B.StopTimer,?,?) ];
   189: [[XIC(H43B.NextMotorOK) XIO(H42D.StopTimer.EN) ,XIC(H42D.HandAuto) ] XIC(H42D.RunStop) XIO(H42D.Fault) OTE(H42D.Run) ,XIC(H42C.StopTimer.DN) TON(H42D.StopTimer,?,?) ];
